# EPICS autosave request: iocBoot/ioc13PECell/Agilent_PS66xxA_settings.req
# FILE... SRS_PS3xx_settings.req
# SRS High Voltage Power Supply
$(P)PS66xxA:$(S):Read.SCAN
